{attribute 'qualified_only'}
{attribute 'strict'}
TYPE E_NCI_CHANNEL_ERROR :
(
  e_Null,
  e_InvalidReference_ChannelRef,
  e_AxisConfigurationMismatch_McAxis,
  e_AxisConfigurationMismatch_AuxAxis


);
END_TYPE

(* stored: Version 1.1.0.1, ProductVersion 3.1.4024.12
   DUT E_NCI_CHANNEL_ERROR: Id {51414efa-601c-064f-30dd-c04a2fdcba9f} *)
